INTERFACE I_Bool

PROPERTY value : BOOL
GET
END_GET
END_PROPERTY

END_INTERFACE

(* stored: Version 1.1.0.1, ProductVersion 3.1.4026.18
   Itf I_Bool: Id {b1a2c3d4-e5f6-7890-abcd-ef1234567890}
   Property value: Id {c2b3d4e5-f6a7-8901-bcde-f12345678901}
   Get Get: Id {d3c4e5f6-a7b8-9012-cdef-123456789012} *)
